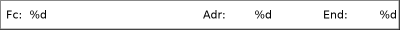
VISUALIZATION VIS_JOB  // 400x30
VAR_INPUT
	ITF_MBJOBIN		:	ITF_MBJOB;
END_VAR
    Frame (0,0 400x30), invisible if: NOT __QUERYINTERFACE(ITF_MBJOBIN,ITF_MBJOBIN)
        shows VIS_JOB_QUERRY(ITF_MBJOBIN := ITF_MBJOBIN)
END_VISUALIZATION

// 40 Visualizations/MBJOB/VIS_JOB_QUERRY
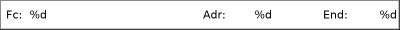
VISUALIZATION VIS_JOB_QUERRY  // 400x30
VAR_INPUT
	ITF_MBJOBIN		:	ITF_MBJOB;
END_VAR
    Rectangle (0,0 400x30)
    Textfield (0,0 25x30), "Fc:"
    Textfield (25,0 25x30), "%d", text variable: ITF_MBJOBIN.byMbFunction
    Textfield (200,0 30x30), "Adr:"
    Textfield (230,0 45x30), "%d", text variable: ITF_MBJOBIN.wMbAdress
    Textfield (320,0 30x30), "End:"
    Textfield (350,0 50x30), "%d", text variable: (ITF_MBJOBIN.wMbAdress + ITF_MBJOBIN.wQuantity-1)
    Rectangle (0,0 400x30)
END_VISUALIZATION

// 40 Visualizations/CLIENTMANAGER/OVERWIEV/VIS_CLIENT_MANAGER_OVERWIEV
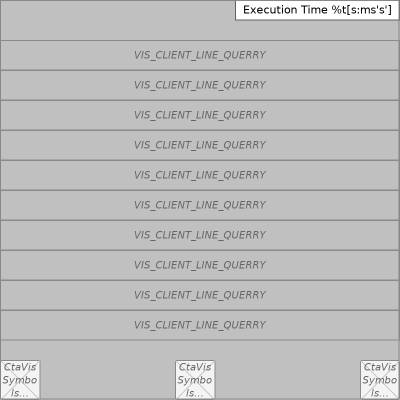
VISUALIZATION VIS_CLIENT_MANAGER_OVERWIEV  // 400x400
VAR_INPUT
	ITF_CLIENT_MANAGER_IN : ITF_MB_CLIENTMANAGER;
END_VAR
    Frame (0,0 400x400), invisible if: NOT __QUERYINTERFACE(ITF_CLIENT_MANAGER_IN,ITF_CLIENT_MANAGER_IN)
        shows VIS_CLIENT_MANAGER_OVERWIEV_QUERRY(ITF_CLIENT_MANAGER_IN := ITF_CLIENT_MANAGER_IN)
END_VISUALIZATION

// 40 Visualizations/CLIENTMANAGER/OVERWIEV/VIS_CLIENT_MANAGER_OVERWIEV_QUERRY
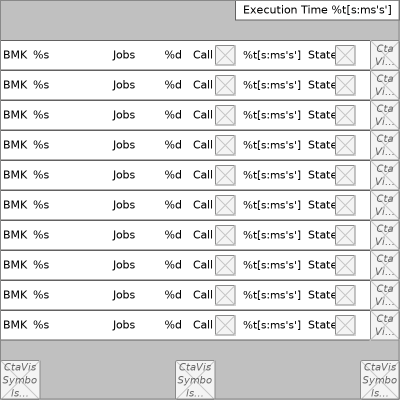
VISUALIZATION VIS_CLIENT_MANAGER_OVERWIEV_QUERRY  // 400x400
VAR_INPUT
	ITF_CLIENT_MANAGER_IN : ITF_MB_CLIENTMANAGER;
END_VAR
    Rectangle (0,0 400x400)
    Image (360,360 40x40), image: CtaVisSymbols.ImagePool.arrow-right_square
        OnMouseClick: execute { ITF_CLIENT_MANAGER_IN.RELOAD_ARRAY(FALSe,TRUE,FALSE); }
    Image (0,360 40x40), image: CtaVisSymbols.ImagePool.arrow-left_square
        OnMouseClick: execute { ITF_CLIENT_MANAGER_IN.RELOAD_ARRAY(FALSe,FALse,TRUE); }
    Image (175,360 40x40), image: CtaVisSymbols.ImagePool.refresh
        OnMouseClick: execute { ITF_CLIENT_MANAGER_IN.RELOAD_ARRAY(TRUE,FALSE,FALSE); }
    Textfield (235,0 165x20), "Execution Time %t[s:ms's']", text variable: ITF_CLIENT_MANAGER_IN.OperationTime
    Frame (0,40 400x300)
        shows VIS_CLIENT_MANAGER_TABLE(AY_ITF_CLIENTS := ITF_CLIENT_MANAGER_IN.AY_ITF_MBCLIENT_VIS)
END_VISUALIZATION

// 40 Visualizations/CLIENTMANAGER/OVERWIEV/VIS_CLIENT_MANAGER_TABLE
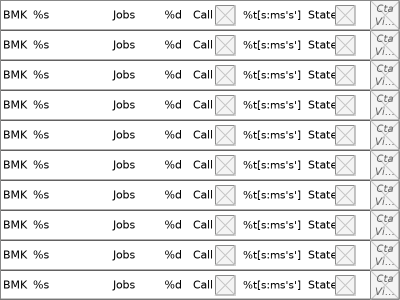
VISUALIZATION VIS_CLIENT_MANAGER_TABLE  // 400x300
VAR_INPUT
	AY_ITF_CLIENTS	:	ARRAY[0..9] OF ITF_CLIENT;
END_VAR
    Frame (0,0 400x30)
        shows VIS_CLIENT_LINE(ITF_CLIENTIN := AY_ITF_CLIENTS[0])
    Frame (0,30 400x30)
        shows VIS_CLIENT_LINE(ITF_CLIENTIN := AY_ITF_CLIENTS[1])
    Frame (0,60 400x30)
        shows VIS_CLIENT_LINE(ITF_CLIENTIN := AY_ITF_CLIENTS[2])
    Frame (0,90 400x30)
        shows VIS_CLIENT_LINE(ITF_CLIENTIN := AY_ITF_CLIENTS[3])
    Frame (0,120 400x30)
        shows VIS_CLIENT_LINE(ITF_CLIENTIN := AY_ITF_CLIENTS[4])
    Frame (0,150 400x30)
        shows VIS_CLIENT_LINE(ITF_CLIENTIN := AY_ITF_CLIENTS[5])
    Frame (0,180 400x30)
        shows VIS_CLIENT_LINE(ITF_CLIENTIN := AY_ITF_CLIENTS[6])
    Frame (0,210 400x30)
        shows VIS_CLIENT_LINE(ITF_CLIENTIN := AY_ITF_CLIENTS[7])
    Frame (0,240 400x30)
        shows VIS_CLIENT_LINE(ITF_CLIENTIN := AY_ITF_CLIENTS[8])
    Frame (0,270 400x30)
        shows VIS_CLIENT_LINE(ITF_CLIENTIN := AY_ITF_CLIENTS[9])
END_VISUALIZATION

// 40 Visualizations/CLIENTMANAGER/PARAMETER/VIS_CLIENT_MANAGER_PARAMETER
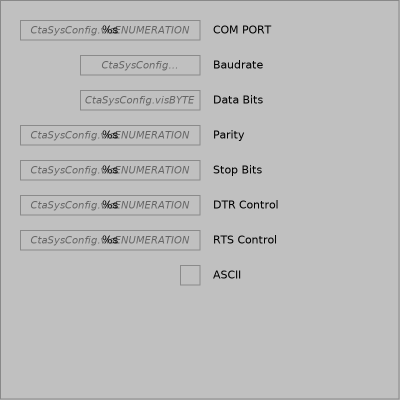
VISUALIZATION VIS_CLIENT_MANAGER_PARAMETER  // 400x400
VAR_INPUT
	ITF_CLIENT_MANAGER_IN : ITF_MB_CLIENTMANAGER;	
END_VAR
    Rectangle (0,0 400x400)
    Frame (0,0 400x400)
        shows VIS_CLIENT_MANAGER_PARAMETER_TCP(ITF_CLIENT_MANAGER_IN := ITF_CLIENT_MANAGER_IN)
    Frame (0,0 400x400)
        shows VIS_CLIENT_MANAGER_PARAMETER_RTU(ITF_CLIENT_MANAGER_IN := ITF_CLIENT_MANAGER_IN)
END_VISUALIZATION

// 40 Visualizations/SERVER/DIA_SERVER
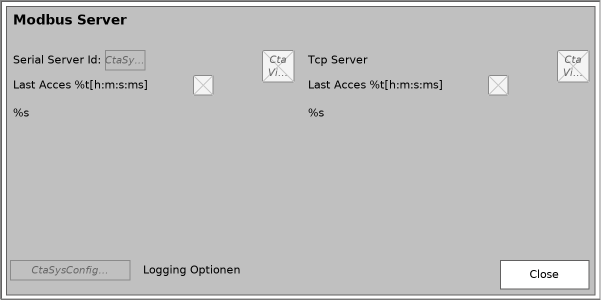
VISUALIZATION DIA_SERVER  // 601x300
VAR_INPUT
	ITF_SERVER_INFO_PARA_IN : ITF_SERVER_INFO_PARA;
END_VAR
    RoundedRectangle (1,1 599x299)
    RoundedRectangle (6,6 589x289)
    RoundedRectangle (500,260 89x29), "Close"
        OnMouseClick:  Dialog=Current Dialog, Result=OK, NumpadKeypadSet=True
    Label (10,5 150x30), "Modbus Server"
    InvisibleInput (1,1 600x40)
    Frame (10,50 285x200)
        shows VIS_SERVER_SERIAL_STATE(ITF_SERVER_INFO_PARA_IN := ITF_SERVER_INFO_PARA_IN)
    Frame (305,50 285x200)
        shows VIS_SERVER_TCP_STATE(ITF_SERVER_INFO_PARA_IN := ITF_SERVER_INFO_PARA_IN)
    Label (140,260 150x20), "Logging Optionen"
    Frame (10,260 120x20)
        shows CtaSysConfig.visDWORD_HEX(visfbDWORDIn := ITF_SERVER_INFO_PARA_IN.P_LoggingOp)
END_VISUALIZATION

// 40 Visualizations/CLIENTMANAGER/RTU/PARAMETER/VIS_CLIENT_MANAGER_PARAMETER_RTU
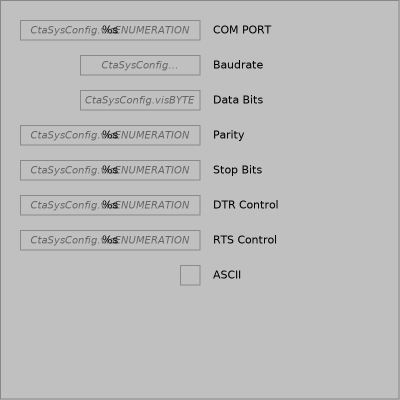
VISUALIZATION VIS_CLIENT_MANAGER_PARAMETER_RTU  // 400x400
VAR_INPUT
	ITF_CLIENT_MANAGER_IN : ITF_MB_CLIENTMANAGER;	
END_VAR
VAR
	ITF_CLIENT_MANAGER_RTU_IN : ITF_MB_CLIENTMANAGER_RTU;	
END_VAR
    Frame (0,0 400x400), invisible if: NOT __QUERYINTERFACE(ITF_CLIENT_MANAGER_IN,ITF_CLIENT_MANAGER_RTU_IN)
        shows VIS_CLIENT_MANAGER_PARAMETER_RTU_TEMP(ITF_CLIENT_MANAGER_RTU_IN := ITF_CLIENT_MANAGER_RTU_IN)
END_VISUALIZATION

// 40 Visualizations/CLIENTMANAGER/RTU/PARAMETER/VIS_CLIENT_MANAGER_PARAMETER_RTU_QUERY
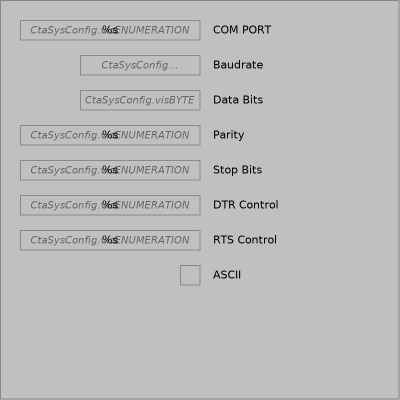
VISUALIZATION VIS_CLIENT_MANAGER_PARAMETER_RTU_QUERY  // 400x400
VAR_INPUT
	ITF_CLIENT_MANAGER_RTU_IN : ITF_MB_CLIENTMANAGER_RTU;	
END_VAR
    Rectangle (0,0 400x400)
    Frame (20,20 180x20), text list: 'TXT_COMPORT', text index: ITF_CLIENT_MANAGER_RTU_IN.P_fbenPort.proValue
        shows CtaSysConfig.visENUMERATION(visfbENUIn := ITF_CLIENT_MANAGER_RTU_IN.P_fbenPort)
    Label (210,20 150x20), "COM PORT"
    Label (210,55 150x20), "Baudrate"
    Frame (80,55 120x20)
        shows CtaSysConfig.visDWORD_DEZ(visfbDWORDIn := ITF_CLIENT_MANAGER_RTU_IN.P_fbdwBaudrate)
    Label (210,90 150x20), "Data Bits"
    Frame (80,90 120x20)
        shows CtaSysConfig.visBYTE(visfbBYTEIn := ITF_CLIENT_MANAGER_RTU_IN.P_fbbyDataBits)
    Label (210,125 150x20), "Parity"
    Frame (20,125 180x20)
        shows CtaSysConfig.visENUMERATION(visfbENUIn := ITF_CLIENT_MANAGER_RTU_IN.P_fbenParity)
    Label (210,160 150x20), "Stop Bits"
    Frame (20,160 180x20)
        shows CtaSysConfig.visENUMERATION(visfbENUIn := ITF_CLIENT_MANAGER_RTU_IN.P_fbenStopBits)
    Label (210,195 150x20), "DTR Control"
    Frame (20,195 180x20)
        shows CtaSysConfig.visENUMERATION(visfbENUIn := ITF_CLIENT_MANAGER_RTU_IN.P_fbenDTRControl)
    Frame (20,230 180x20)
        shows CtaSysConfig.visENUMERATION(visfbENUIn := ITF_CLIENT_MANAGER_RTU_IN.P_fbenRTSControl)
    Label (210,230 150x20), "RTS Control"
    Frame (180,265 20x20)
        shows CtaSysConfig.visBOOL(visfbBOOLIn := ITF_CLIENT_MANAGER_RTU_IN.P_fbxRtuAscii)
    Label (210,265 150x20), "ASCII"
    Textfield (40,20 140x20), "%s", text list: 'TXT_COMPORT', text index: ITF_CLIENT_MANAGER_RTU_IN.P_fbenPort.proValue
    Textfield (40,125 140x20), "%s", text list: 'TEXT_PARITY', text index: ITF_CLIENT_MANAGER_RTU_IN.P_fbenParity.proValue
    Textfield (40,160 140x20), "%s", text list: 'TEXT_STOPBITS', text index: ITF_CLIENT_MANAGER_RTU_IN.P_fbenStopBits.proValue
    Textfield (40,195 140x20), "%s", text list: 'TEXT_DTR_CONTROL', text index: ITF_CLIENT_MANAGER_RTU_IN.P_fbenDTRControl.proValue
    Textfield (40,230 140x20), "%s", text list: 'TEXT_RTS_CONTROL', text index: ITF_CLIENT_MANAGER_RTU_IN.P_fbenRTSControl.proValue
END_VISUALIZATION

// 40 Visualizations/CLIENTMANAGER/RTU/PARAMETER/VIS_CLIENT_MANAGER_PARAMETER_RTU_TEMP
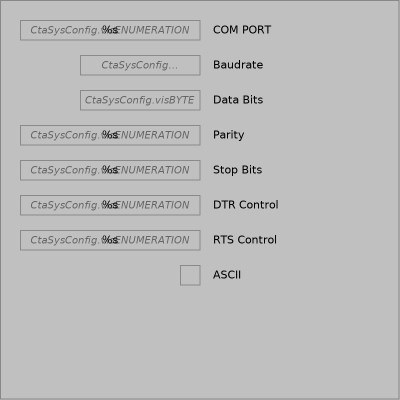
VISUALIZATION VIS_CLIENT_MANAGER_PARAMETER_RTU_TEMP  // 400x400
VAR_INPUT
	ITF_CLIENT_MANAGER_RTU_IN : ITF_MB_CLIENTMANAGER_RTU;	
END_VAR
    Frame (0,0 400x400), invisible if: NOT __QUERYINTERFACE(ITF_CLIENT_MANAGER_RTU_IN,ITF_CLIENT_MANAGER_RTU_IN)
        shows VIS_CLIENT_MANAGER_PARAMETER_RTU_QUERY(ITF_CLIENT_MANAGER_RTU_IN := ITF_CLIENT_MANAGER_RTU_IN)
END_VISUALIZATION

// 40 Visualizations/SERVER/SERIAL/PARAMETER/DIA_SERVER_SERIAL_PARAMETER
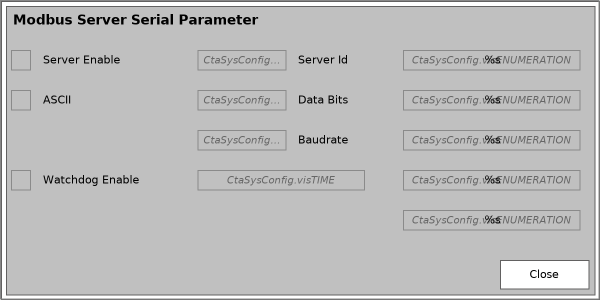
VISUALIZATION DIA_SERVER_SERIAL_PARAMETER  // 600x300
VAR_INPUT
	ITF_SERVER_INFO_PARA_IN : ITF_SERVER_INFO_PARA;
END_VAR
    RoundedRectangle (1,1 599x299)
    RoundedRectangle (6,6 589x289)
    RoundedRectangle (500,260 89x29), "Close"
        OnMouseClick:  Dialog=Current Dialog, Result=OK, NumpadKeypadSet=True
    Label (10,5 210x30), "Modbus Server Serial Parameter"
    InvisibleInput (0,0 600x40)
    Frame (11,50 579x200), invisible if: NOT __QUERYINTERFACE(ITF_SERVER_INFO_PARA_IN,ITF_SERVER_INFO_PARA_IN)
        shows VIS_SERVER_SERIAL_PARAMETER(ITF_SERVER_INFO_PARA_IN := ITF_SERVER_INFO_PARA_IN)
END_VISUALIZATION

// 40 Visualizations/SERVER/SERIAL/PARAMETER/VIS_SERVER_SERIAL_PARAMETER
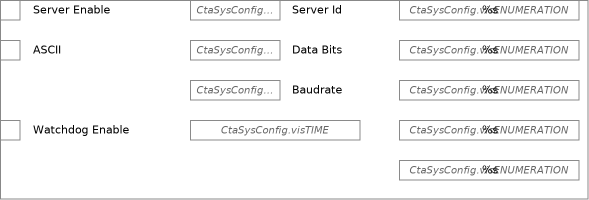
VISUALIZATION VIS_SERVER_SERIAL_PARAMETER  // 589x200
VAR_INPUT
	ITF_SERVER_INFO_PARA_IN : ITF_SERVER_INFO_PARA;
END_VAR
    Frame (0,0 20x20)
        shows CtaSysConfig.visBOOL(visfbBOOLIn := ITF_SERVER_INFO_PARA_IN.P_Serial_fbxEnable)
    Label (30,0 140x20), "Server Enable"
    Frame (399,0 180x20)
        shows CtaSysConfig.visENUMERATION(visfbENUIn := ITF_SERVER_INFO_PARA_IN.P_Serial_fbenPort)
    Label (289,0 100x20), "Server Id"
    Frame (190,0 90x20)
        shows CtaSysConfig.visUSINT(visfbUSINTIn := ITF_SERVER_INFO_PARA_IN.P_Serial_fbusiNodeId)
    Frame (399,40 180x20)
        shows CtaSysConfig.visENUMERATION(visfbENUIn := ITF_SERVER_INFO_PARA_IN.P_Serial_fbenParity)
    Frame (399,80 180x20)
        shows CtaSysConfig.visENUMERATION(visfbENUIn := ITF_SERVER_INFO_PARA_IN.P_Serial_fbenStopBits)
    Frame (399,120 180x20)
        shows CtaSysConfig.visENUMERATION(visfbENUIn := ITF_SERVER_INFO_PARA_IN.P_Serial_fbenDTRControl)
    Frame (399,160 180x20)
        shows CtaSysConfig.visENUMERATION(visfbENUIn := ITF_SERVER_INFO_PARA_IN.P_Serial_fbenRTSControl)
    Frame (190,40 90x20)
        shows CtaSysConfig.visBYTE(visfbBYTEIn := ITF_SERVER_INFO_PARA_IN.P_Serial_fbbyDataBits)
    Label (289,40 100x20), "Data Bits"
    Label (289,80 100x20), "Baudrate"
    Frame (190,80 90x20)
        shows CtaSysConfig.visDWORD_DEZ(visfbDWORDIn := ITF_SERVER_INFO_PARA_IN.P_Serial_fbdwBaudrate)
    Frame (0,120 20x20)
        shows CtaSysConfig.visBOOL(visfbBOOLIn := ITF_SERVER_INFO_PARA_IN.P_Serial_fbxEnableWatchDog)
    Label (30,120 140x20), "Watchdog Enable"
    Label (30,40 140x20), "ASCII"
    Frame (0,40 20x20)
        shows CtaSysConfig.visBOOL(visfbBOOLIn := ITF_SERVER_INFO_PARA_IN.P_Serial_fbxRtuAscii)
    Frame (190,120 170x20)
        shows CtaSysConfig.visTIME(visfbTIMEIn := ITF_SERVER_INFO_PARA_IN.P_Serial_fbtWatchDog)
    Textfield (420,160 140x20), "%s", text list: 'TEXT_RTS_CONTROL', text index: ITF_SERVER_INFO_PARA_IN.P_Serial_fbenRTSControl.proValue
    Textfield (420,120 140x20), "%s", text list: 'TEXT_DTR_CONTROL', text index: ITF_SERVER_INFO_PARA_IN.P_Serial_fbenDTRControl.proValue
    Textfield (420,80 140x20), "%s", text list: 'TEXT_STOPBITS', text index: ITF_SERVER_INFO_PARA_IN.P_Serial_fbenStopBits.proValue
    Textfield (420,40 140x20), "%s", text list: 'TEXT_PARITY', text index: ITF_SERVER_INFO_PARA_IN.P_Serial_fbenParity.proValue
    Textfield (420,0 140x20), "%s", text list: 'TXT_COMPORT', text index: ITF_SERVER_INFO_PARA_IN.P_Serial_fbenPort.proValue
END_VISUALIZATION

// 40 Visualizations/SERVER/TCP/VIS_SERVER_TCP_STATE
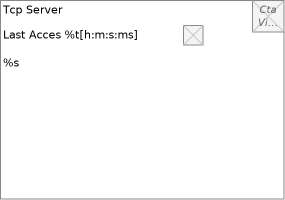
VISUALIZATION VIS_SERVER_TCP_STATE  // 285x200
VAR_INPUT
	ITF_SERVER_INFO_PARA_IN : ITF_SERVER_INFO_PARA;
END_VAR
    Frame (0,0 285x200), invisible if: NOT __QUERYINTERFACE(ITF_SERVER_INFO_PARA_IN,ITF_SERVER_INFO_PARA_IN)
        shows VIS_SERVER_TCP_STATE_INFO(ITF_SERVER_INFO_PARA_IN := ITF_SERVER_INFO_PARA_IN)
END_VISUALIZATION

// 40 Visualizations/SERVER/TCP/VIS_SERVER_TCP_STATE_INFO
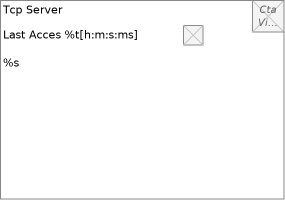
VISUALIZATION VIS_SERVER_TCP_STATE_INFO  // 285x200
VAR_INPUT
	ITF_SERVER_INFO_PARA_IN : ITF_SERVER_INFO_PARA;
END_VAR
    Label (0,0 96x20), "Tcp Server"
    Textfield (0,55 285x144), "%s", text variable: ITF_SERVER_INFO_PARA_IN.RequestDataTcp
    Textfield (0,25 178x20), "Last Acces %t[h:m:s:ms]", text variable: ITF_SERVER_INFO_PARA_IN.NoTcpAccesSince
    Image (183,25 20x20), invisible if: NOT ITF_SERVER_INFO_PARA_IN.TimeOutTcpWatchDog, image: CtaVisSymbols.ImagePool.CtaError
    Image (252,0 32x32), image: CtaVisSymbols.ImagePool.gear
        OnMouseClick:  Dialog=DIA_SERVER_TCP_PARAMETER, Parameters={ITF_SERVER_INFO_PARA_IN: ITF_SERVER_INFO_PARA_IN}, OpenCentered=True
END_VISUALIZATION

// 40 Visualizations/SERVER/TCP/PARAMETER/DIA_SERVER_TCP_PARAMETER
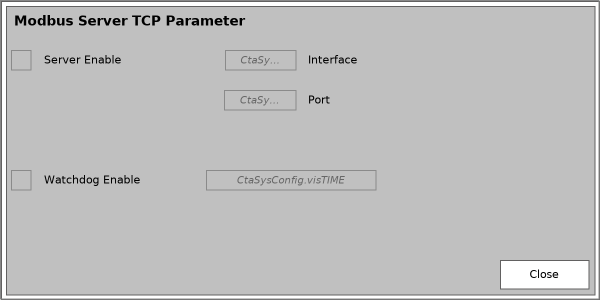
VISUALIZATION DIA_SERVER_TCP_PARAMETER  // 600x300
VAR_INPUT
	ITF_SERVER_INFO_PARA_IN : ITF_SERVER_INFO_PARA;
END_VAR
    RoundedRectangle (1,1 599x299)
    RoundedRectangle (6,6 589x289)
    RoundedRectangle (500,260 89x29), "Close"
        OnMouseClick:  Dialog=Current Dialog, Result=OK, NumpadKeypadSet=True
    Label (11,6 210x30), "Modbus Server TCP Parameter"
    InvisibleInput (0,0 600x40)
    Frame (11,50 579x200), invisible if: NOT __QUERYINTERFACE(ITF_SERVER_INFO_PARA_IN,ITF_SERVER_INFO_PARA_IN)
        shows VIS_SERVER_TCP_PARAMETER(ITF_SERVER_INFO_PARA_IN := ITF_SERVER_INFO_PARA_IN)
END_VISUALIZATION

// 40 Visualizations/SERVER/TCP/PARAMETER/VIS_SERVER_TCP_PARAMETER
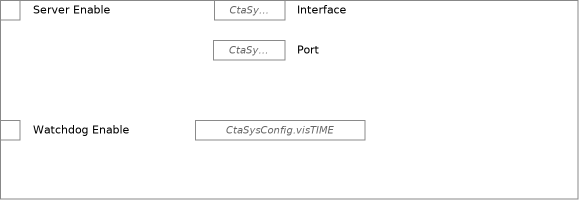
VISUALIZATION VIS_SERVER_TCP_PARAMETER  // 579x200
VAR_INPUT
	ITF_SERVER_INFO_PARA_IN : ITF_SERVER_INFO_PARA;
END_VAR
    Frame (0,0 20x20)
        shows CtaSysConfig.visBOOL(visfbBOOLIn := ITF_SERVER_INFO_PARA_IN.P_Tcp_fbxEnable)
    Label (30,0 140x20), "Server Enable"
    Label (294,0 100x20), "Interface"
    Label (294,40 100x20), "Port"
    Frame (0,120 20x20)
        shows CtaSysConfig.visBOOL(visfbBOOLIn := ITF_SERVER_INFO_PARA_IN.P_Tcp_fbxEnableWatchDog)
    Label (30,120 140x20), "Watchdog Enable"
    Frame (195,120 170x20)
        shows CtaSysConfig.visTIME(visfbTIMEIn := ITF_SERVER_INFO_PARA_IN.P_Tcp_fbtWatchDog)
    Frame (214,0 71x20)
        shows CtaSysConfig.visSTRING40(visfbSTRING40In := ITF_SERVER_INFO_PARA_IN.P_Tcp_fbstInterface)
    Frame (213,40 72x20)
        shows CtaSysConfig.visWORD_DEZ(visfbWORDIn := ITF_SERVER_INFO_PARA_IN.P_Tcp_fbwPort)
END_VISUALIZATION

(* text list TEXT_DTR_CONTROL (id | default)
  0 | DTR Disable
  1 | DTR Enable
  2 | DTR Handshake
   |  *)

(* text list TEXT_PARITY (id | default)
  0 | None
  1 | Odd
  2 | Even
   |  *)

(* text list TEXT_RTS_CONTROL (id | default)
  0 | RTS Disable
  1 | RTS Enable
  2 | RTS Handshake
  3 | RTS Toggle
   |  *)

(* text list TEXT_STOPBITS (id | default)
  1 | ONE
  2 | ONE DOT FIVE
  3 | TWO
   |  *)

(* text list TXT_COMPORT (id | default)
  0 | NO COM
  1 | COM1
  2 | COM2
  3 | COM3
  4 | COM4
  5 | COM5
  6 | COM6
  7 | COM7
  8 | COM8
  9 | COM9
  10 | COM10
   |  *)

(* text list txtHandshake (id | default)
  0 | Default
  1 | None
  2 | XON XOFF
  3 | DTE RTS CTS
  4 | DCE RTS CTS
  5 | DTE DSR DTR
  6 | DCE DSR DTR
  7 | RTS Lead Time
   |  *)

(* text list txtParity (id | default)
  0 | Default
  1 | None
  2 | Odd
  3 | Even
  4 | Mark
  5 | Space
   |  *)

(* text list txtPhysikalLayer (id | default)
  0 | Default
  1 | RS232
  2 | RS422
  3 | RS423
  4 | RS485 half duplex
  5 | RS485 full duplex
  6 | DMX half duplex
   |  *)

(* text list txtStopBits (id | default)
  0 | Default
  1 | None
  2 | Minimum
  3 | One
  4 | OneDotFive
  5 | Two
  255 | Maximum
   |  *)

(* text list txtLoggingOp (id | default)
  0 | Name	Initial	Comment / None /  / 16#0	  / Init /  / 16#1	Initialization / ServerStartStop /  / 16#2	Start / stop of server / ServerDataModel /  / 16#4	Server data model information / ServerException /  / 16#8	Server rejected requests with exception / ServerExceptionReason /  / 16#10	Server rejected requests with exception, detailed reason / ServerReceivedValidRequests /  / 16#20	Server received valid request / ServerRequestDetails /  / 16#40	Server received request - details / ClientConnectDisconnect /  / 16#80	Client connect / disconnect. / ClientReceivedValidReplies /  / 16#100	Client received valid reply / ClientReplyDetails /  / 16#200	Client received valid reply - details / ClientRequestStateChange /  / 16#400	ClientRequest state changes / SendFrames /  / 16#800	Send frame / WarnOnReceivedInvalidFrames /  / 16#1000	Warn on invalid frames received / ClientTcpSocket /  / 16#2000	Log ClientTcp socket activities / ServerTcpSocket /  / 16#4000	Log ServerTcp socket activities / SysComOpenClose /  / 16#8000	Log SysCom open/close / Internals /  / 16#10000	  / SysComHandlerStateChange /  / 16#20000	Log SysComHandler state changes / All /  / 16#FFFFFFFF	 
   |  *)
